INTERFACE DemandedSpeedInterface

METHOD GetSpeed : UINT
END_METHOD

END_INTERFACE

(* stored: Version 1.1.0.1, ProductVersion 3.1.4022.16
   Itf DemandedSpeedInterface: Id {a53454b6-6512-444b-84d7-3c5467799a66}
   Method GetSpeed: Id {b05dbdd3-659d-45cb-acd6-5f0a0bcfc42e} *)
